// TIA Portal V20 export
TYPE "OPC_DestInfo_Ack"
// stored: Namespace ProductionLine
   STRUCT
      AckSeq : Int;   // //Communication flag, described in the Data tab
   END_STRUCT;
END_TYPE
